GLOBALCONSTANTS DefaultPool_Dreieck_PositionMarker (* Position marker constants (child/parent object IDs, travel bounds, center offset) *)
  PACKAGE Uebungen::const::UT::Dreieck;
  VAR_GLOBAL CONSTANT
    Container_PositionMarker : isobus::utils::childposition::PositionMarker_S := (u16ChildId := 16000, u16ParentId := 3000, r32MinPos := 0.0, r32MaxPos := 84.0, r32Center := 42.0, s16YPosition := 0);
  END_VAR
END_GLOBALCONSTANTS
